//LREAL Slew rate limitter with a timebased change rate
FUNCTION_BLOCK SlewRateLimitter
VAR_INPUT
	IN														: LREAL := 0.0;	 //Actual value
	Sync													: BOOL := FALSE; //Sync signal sets IN to Q	
	Cycletime												: LREAL := 0.001; //cycletime in ms
	Rate													: LREAL := 1.0;	 // changes per second
END_VAR                 									
VAR_OUTPUT              									
	Q														: LREAL := 0.0;   //Output
END_VAR                 									
VAR                     	
	x														: LREAL := 0.0;
END_VAR

//Based on MC_AxUtiSlewRateLimitter_BkPlcMc from TcPlcLibHydraulics , Author WOs
IF Cycletime <= 0.0001 OR Rate <= 0.0 OR Sync
THEN
	Q														:= IN;
ELSE                    									
	x														:= Cycletime * Rate;
	IF ABS(IN) > X OR ABS(Q > In)
	THEN //Start ramping only after In is greater than Rate and as long as Q is greater (if In jumps to zero)
		Q													:= Q + LIMIT(-x , IN - Q , x); 		
	ELSE
		Q													:= In;
	END_IF
END_IF

METHOD PUBLIC synchronize : BOOL //Return value = TRUE if execution finished
VAR_INPUT
	IN														:	LREAL;
END_VAR
Q 															:= IN;
Synchronize 												:= TRUE;
END_METHOD

END_FUNCTION_BLOCK

(* stored: Version 1.1.0.1, ProductVersion 3.1.4024.9
   POU SlewRateLimitter: Id {69b14dad-ebaa-4236-9ab3-2cefa783c1e1}, SpecialFunc None
   Method synchronize: Id {2b3fd695-89db-44b9-938c-b96cee39fdd6} *)
